{attribute 'qualified_only'}
VAR_GLOBAL
	K1 :BOOL; // Vereinzelner
	K2 :BOOL; // Füllen
	P1 :BOOL; // Behälter leer
	Q1 :BOOL; // Förderband
END_VAR

(* stored: Version 1.1.0.1, ProductVersion 3.1.4024.5
   GVL SimDA: Id {efa3d63a-96e1-4204-b1e7-9f3703bd4f03} *)
